// TIA Portal V21 export
DATA_BLOCK "MacchinaARicetta"   // DB20
{ S7_Optimized_Access := 'TRUE' }
// stored: MemoryReserve 100
   VAR RETAIN
      "M" : Array[0.."K_NumMacchinaARicetta"] of "Std_RicettaUniverale";
   END_VAR
   VAR
      Hmi_Custom : Struct   // Struttura solo per questa macchina
         Spiedinatrice : Struct
            GeneraQuoteMotore : Bool := FALSE;
            CalcolaCicliTaglio : Bool := FALSE;
         END_STRUCT;
      END_STRUCT;
   END_VAR
BEGIN
   "M"[0].Lavoro.NomeFormato := '';
   "M"[0].Lavoro.DatoReal[0..10] := 0.0;
   "M"[0].Lavoro.DatoBool[0..10] := FALSE;
   "M"[0].Modifica.NomeFormato := '';
   "M"[0].Modifica.DatoReal[0..10] := 0.0;
   "M"[0].Modifica.DatoBool[0..10] := FALSE;
   "M"[0].Originali.NomeFormato := '';
   "M"[0].Originali.DatoReal[0..10] := 0.0;
   "M"[0].Originali.DatoBool[0..10] := FALSE;
   "M"[0].Archivio[0].NomeFormato := '';
   "M"[0].Archivio[0].DatoReal[0..10] := 0.0;
   "M"[0].Archivio[0].DatoBool[0..10] := FALSE;
   "M"[0].Hmi.NumDatoRicettaBool := 0;
   "M"[0].Hmi.NumDatoRicettaReal := 0;
   "M"[0].Hmi.CodiceMacchinario := 0;
   "M"[0].Hmi.Indice_Selezionata := 0;
   "M"[0].Hmi.Indice_RicettaAttuale := 0;
   "M"[0].Hmi.Indice_CopiaDa := 0;
   "M"[0].Hmi.Indice_CopiaIn := 0;
   "M"[0].Hmi.Esegui_Annulla := FALSE;
   "M"[0].Hmi.Esegui_Carica := FALSE;
   "M"[0].Hmi.Esegui_Salva := FALSE;
   "M"[0].Hmi.Esegui_Copia := FALSE;
   "M"[0].Hmi.Esegui_ModificaRicettaInLavoro := FALSE;
   "M"[0].Hmi.Esegui_ModificaRicettaInArchivio := FALSE;
   "M"[0].Hmi.InCorso_ModificaRicettaInLavoro := FALSE;
   "M"[0].Hmi.InCorso_ModificaRicettaInArchivio := FALSE;
   "M"[0].Hmi.Scelta_CopiaDa := FALSE;
   "M"[0].Hmi.Scelta_CopiaIn := FALSE;
   "M"[0].Hmi.RichiediSalvataggio := FALSE;
   "M"[0].Hmi.FocusArchivio := FALSE;
   "M"[0].Hmi.AvviaCopia := FALSE;
   "M"[0].Hmi.AbilitaCarica := FALSE;
   "M"[0].Hmi.AbilitaCopia := FALSE;
   "M"[0].Hmi.Abilita_ModificaRicettaInLavoro := FALSE;
   "M"[0].Hmi.Abilita_ModificaRicettaInArchivio := FALSE;
   "M"[0].Hmi.MemoOldSelezione := 0;
   "M"[0].Hmi.MostraOriginali := FALSE;
   "M"[0].Hmi.Archivio.AbilitaIncrementoRicetta := FALSE;
   "M"[0].Hmi.Archivio.AbilitaDecrementoRicetta := FALSE;
   "M"[0].Hmi.Archivio.IndiceFormatoVisualizzato := 0;
   "M"[0].Hmi.Archivio.IndiceHmi[0..5] := 0;
   "M"[0].Hmi.Archivio.NomeHmi[0..5] := '';
   "M"[0].Hmi.Archivio.SelezioneHmi[0..5] := FALSE;
   "M"[0].Out.ScriviDatiLagica := FALSE;
   "M"[0].Allarmi."A"[0..2].Abilitato := FALSE;
   "M"[0].Allarmi."A"[0..2].Stato := FALSE;
   "M"[0].Allarmi."A"[0..2].Silenziato := FALSE;
   "M"[0].Allarmi."A"[0..2].EnWarnHmi := FALSE;
   "M"[0].Allarmi."A"[0..2].EnCadutaCiclo := FALSE;
   "M"[0].Allarmi.WordHMI := 16#0000;
END_DATA_BLOCK
